// TwinCAT 3 PLC project core_test
// ProgramVersion: 3.1.4026.16
// libraries:
//   [Nepionic Core], * (Nepionic)
//   Tc2_Standard, * (Beckhoff Automation GmbH)
//   Tc2_System, * (Beckhoff Automation GmbH)
// project tree:
//   Tests/ Test.TcPOU
//   Tasks/ PlcTask.TcTTO
// real-time tasks:
//   TASK PlcTask: cycle T#10ms, priority 20, ADS port 350

CONFIGURATION core_test
    RESOURCE PLC ON TwinCAT3
        TASK PlcTask(INTERVAL := T#10ms, PRIORITY := 20);
        PROGRAM Test WITH PlcTask : Test;
    END_RESOURCE
END_CONFIGURATION

// ---- Tests/Test.TcPOU
PROGRAM Test
VAR
END_VAR

END_PROGRAM
